Yaskawa INFORM job: pipe_bracket_cylinder_program.JBI

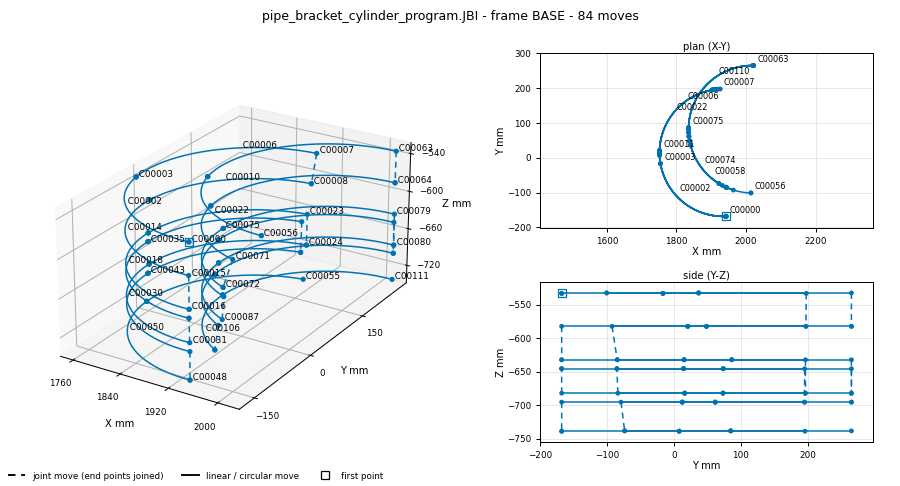
[picture p0: tool path of pipe_bracket_cylinder_program.JBI in frame BASE, 84 of 117 moves have a stored position in this frame; points joined in program order, loops and branches not executed]
/JOB
//NAME pipe_bracket_cylinder_program
//POS
///NPOS 112,0,112,0,0,0
///TOOL 0
///POSTYPE BASE
///RECTAN
///RCONF 0,0,0,0,0,0,0,0,0,0,0,0,0,0,0,0,0,0,0,0,0,0,0,0
C00000=1942.537957,-168.012753,-532.924500,-87.433791,-89.999999,5.000000
C00001=1942.537957,-168.012753,-532.924500,-87.433791,-89.999999,5.000000
C00002=1797.443653,-106.704534,-532.924500,-138.378261,-89.999999,5.000000
C00003=1753.930524,-16.502665,-532.924500,-170.116676,-89.999999,5.000000
C00004=1753.930524,-16.502665,-532.924500,-170.116676,-89.999999,5.000000
C00005=1753.930524,-16.502665,-532.924500,-170.116676,-89.999999,5.000000
C00006=1819.648743,157.692613,-532.924500,128.776952,-90.000000,5.000000
C00007=1925.886728,197.860249,-532.924500,92.645366,-90.000000,5.000000
C00008=1918.014662,197.326376,-582.169500,95.114199,-89.999999,5.000000
C00009=1918.014662,197.326376,-582.169500,95.114199,-89.999999,5.000000
C00010=1800.257643,139.658655,-582.169500,137.069440,-90.000000,5.000000
C00011=1751.301252,20.620145,-582.169500,175.000000,-89.999999,5.000000
C00012=1751.301252,20.620145,-582.169500,175.000000,-89.999999,5.000000
C00013=1751.301252,20.620145,-582.169500,175.000000,-89.999999,5.000000
C00014=1782.935371,-88.085662,-582.169500,-145.768544,-90.000000,5.000000
C00015=1941.730148,-168.047171,-582.169500,-87.686765,-90.000000,5.000000
C00016=1941.975553,-168.037093,-632.172000,-87.609919,-89.999999,5.000000
C00017=1941.975553,-168.037093,-632.172000,-87.609919,-89.999999,5.000000
C00018=1783.333373,-88.668199,-632.172000,-145.547804,-90.000000,5.000000
C00019=1751.212998,15.190866,-632.172000,175.000000,-90.000000,5.000000
C00020=1751.212998,15.190866,-632.172000,175.000000,-90.000000,5.000000
C00021=1751.212998,15.190866,-632.172000,175.000000,-90.000000,5.000000
C00022=1789.567117,127.073517,-632.172000,142.237662,-90.000000,5.000000
C00023=1912.126975,196.703354,-632.172000,96.966683,-90.000000,5.000000
C00024=1911.336404,196.605005,-682.155000,97.215941,-90.000000,5.000000
C00025=1911.336404,196.605005,-682.155000,97.215941,-90.000000,5.000000
C00026=1789.008166,126.348204,-682.155000,142.524163,-90.000000,5.000000
C00027=1751.215641,15.947385,-682.155000,175.000000,-90.000000,5.000000
C00028=1751.215641,15.947385,-682.155000,175.000000,-90.000000,5.000000
C00029=1751.215641,15.947385,-682.155000,175.000000,-90.000000,5.000000
C00030=1786.192815,-92.717556,-682.155000,-143.996770,-90.000000,5.000000
C00031=1942.358131,-168.020724,-682.155000,-87.490110,-90.000000,5.000000
C00032=1941.526633,-168.055278,-645.556460,-175.000000,-60.000000,92.249509
C00033=1941.526633,-168.055278,-645.556460,-175.000000,-60.000000,92.249509
C00034=1780.853143,-84.956813,-645.556460,175.000000,-60.000000,33.055529
C00035=1751.213846,14.313901,-645.556460,-175.000000,-60.000000,5.000000
C00036=1751.213846,14.313901,-645.556460,-175.000000,-60.000000,5.000000
C00037=1751.213846,14.313901,-645.556460,-175.000000,-60.000000,5.000000
C00038=1788.892614,126.197321,-645.556460,175.000000,-60.000000,-37.416375
C00039=1903.454355,195.432275,-645.556460,175.000000,-60.000000,-80.290608
C00040=1902.349178,195.239691,-695.542960,175.000000,-60.000000,-79.939613
C00041=1902.349178,195.239691,-695.542960,175.000000,-60.000000,-79.939613
C00042=1788.632983,125.857115,-695.542960,175.000000,-60.000000,-37.282477
C00043=1751.229898,12.427988,-695.542960,175.000000,-60.000000,5.000000
C00044=1751.229898,12.427988,-695.542960,175.000000,-60.000000,5.000000
C00045=1751.229898,12.427988,-695.542960,175.000000,-60.000000,5.000000
C00046=1782.456963,-87.379003,-695.542960,-175.000000,-60.000000,33.964456
C00047=1942.452445,-168.016565,-695.542960,175.000000,-60.000000,92.539427
C00048=1942.174784,-168.028668,-739.049960,-175.000000,-60.000000,92.452471
C00049=1942.174784,-168.028668,-739.049960,-175.000000,-60.000000,92.452471
C00050=1781.503320,-85.948835,-739.049960,175.000000,-60.000000,33.426633
C00051=1751.353161,7.761270,-739.049960,175.000000,-60.000000,5.000000
C00052=1751.353161,7.761270,-739.049960,175.000000,-60.000000,5.000000
C00053=1751.353161,7.761270,-739.049960,175.000000,-60.000000,5.000000
C00054=1784.506338,120.216512,-739.049960,175.000000,-60.000000,-35.095663
C00055=1906.907155,195.989172,-739.049960,-175.000000,-60.000000,-81.384886
C00056=2014.143483,-100.766826,-532.230000,-91.168935,-89.999999,5.000000
C00057=2014.143483,-100.766826,-532.230000,-91.168935,-89.999999,5.000000
C00058=1899.462167,-57.366095,-532.230000,-130.289001,-89.999999,5.000000
C00059=1840.487082,36.855691,-532.230000,-165.624641,-90.000000,5.000000
C00060=1840.487082,36.855691,-532.230000,-165.624641,-90.000000,5.000000
C00061=1840.487082,36.855691,-532.230000,-165.624641,-90.000000,5.000000
C00062=1900.582124,222.949781,-532.230000,129.831172,-90.000000,5.000000
C00063=2020.961875,265.420918,-532.230000,89.035494,-90.000000,5.000000
C00064=2020.657830,265.425784,-582.179500,89.130635,-89.999999,5.000000
C00065=2020.657830,265.425784,-582.179500,89.130635,-89.999999,5.000000
C00066=1885.350173,208.697868,-582.179500,136.361231,-89.999999,5.000000
C00067=1837.891489,48.564816,-582.179500,-169.377752,-90.000000,5.000000
C00068=1837.891489,48.564816,-582.179500,-169.377752,-90.000000,5.000000
C00069=1837.891489,48.564816,-582.179500,-169.377752,-90.000000,5.000000
C00070=1881.544380,-39.940562,-582.179500,-138.115094,-90.000000,5.000000
C00071=1963.739611,-92.618991,-582.179500,-107.196037,-90.000000,5.000000
C00072=1943.237520,-84.902532,-632.168500,-114.054049,-90.000000,5.000000
C00073=1943.237520,-84.902532,-632.168500,-114.054049,-90.000000,5.000000
C00074=1870.633273,-26.553727,-632.168500,-143.520535,-90.000000,5.000000
C00075=1834.799732,86.439422,-632.168500,175.000000,-90.000000,5.000000
C00076=1834.799732,86.439422,-632.168500,175.000000,-90.000000,5.000000
C00077=1834.799732,86.439422,-632.168500,175.000000,-90.000000,5.000000
C00078=1900.762842,223.100320,-632.168500,129.757582,-90.000000,5.000000
C00079=2021.100654,265.418529,-632.168500,88.992067,-89.999999,5.000000
C00080=2021.557535,265.409920,-682.170500,88.849094,-89.999999,5.000000
C00081=2021.557535,265.409920,-682.170500,88.849094,-89.999999,5.000000
C00082=1881.209361,204.207875,-682.170500,138.272336,-90.000000,5.000000
C00083=1834.977558,73.263237,-682.170500,-175.000000,-90.000000,5.000000
C00084=1834.977558,73.263237,-682.170500,-175.000000,-90.000000,5.000000
C00085=1834.977558,73.263237,-682.170500,-175.000000,-90.000000,5.000000
C00086=1869.380160,-24.838246,-682.170500,-144.185220,-89.999999,5.000000
C00087=1941.074160,-83.920016,-682.170500,-114.797455,-89.999999,5.000000
C00088=1944.487882,-85.455056,-645.550960,-175.000000,-60.000000,66.373654
C00089=1944.487882,-85.455056,-645.550960,-175.000000,-60.000000,66.373654
C00090=1872.022822,-28.408340,-645.550960,175.000000,-60.000000,37.204536
C00091=1834.960316,73.618385,-645.550960,175.000000,-60.000000,5.000000
C00092=1834.960316,73.618385,-645.550960,175.000000,-60.000000,5.000000
C00093=1834.960316,73.618385,-645.550960,175.000000,-60.000000,5.000000
C00094=1893.701616,216.912919,-645.550960,175.000000,-60.000000,-47.304641
C00095=2020.753432,265.424308,-645.550960,175.000000,-60.000000,-90.899280
C00096=2021.249895,265.415842,-695.548960,175.000000,-60.000000,-91.054635
C00097=2021.249895,265.415842,-695.548960,175.000000,-60.000000,-91.054635
C00098=1880.467269,203.370643,-695.548960,-175.000000,-60.000000,-41.377625
C00099=1835.921192,61.673045,-695.548960,175.000000,-60.000000,6.474015
C00100=1835.921192,61.673045,-695.548960,175.000000,-60.000000,6.474015
C00101=1835.921192,61.673045,-695.548960,175.000000,-60.000000,6.474015
C00102=1874.105058,-31.098868,-695.548960,175.000000,-60.000000,38.269005
C00103=1931.752214,-79.287259,-695.548960,-175.000000,-60.000000,61.945168
C00104=1922.138759,-73.784261,-738.575460,175.000000,-60.000000,58.478885
C00105=1922.138759,-73.784261,-738.575460,175.000000,-60.000000,58.478885
C00106=1874.782710,-31.952642,-738.575460,175.000000,-60.000000,38.610046
C00107=1834.769699,84.763058,-738.575460,-175.000000,-60.000000,-5.000000
C00108=1834.769699,84.763058,-738.575460,-175.000000,-60.000000,-5.000000
C00109=1834.769699,84.763058,-738.575460,-175.000000,-60.000000,-5.000000
C00110=1910.745399,230.838368,-738.575460,175.000000,-60.000000,-54.194979
C00111=2020.675033,265.425522,-738.575460,175.000000,-60.000000,-90.874748
///POSTYPE PULSE
///PULSE
EX00000=95232.0
EX00001=275456.0
///POSTYPE PULSE
///PULSE
EC00000=95232.0
EC00001=95232.0
EC00002=95232.0
EC00003=95232.0
EC00004=95232.0
EC00005=95232.0
EC00006=95232.0
EC00007=95232.0
EC00008=95232.0
EC00009=95232.0
EC00010=95232.0
EC00011=95232.0
EC00012=95232.0
EC00013=95232.0
EC00014=95232.0
EC00015=95232.0
EC00016=95232.0
EC00017=95232.0
EC00018=95232.0
EC00019=95232.0
EC00020=95232.0
EC00021=95232.0
EC00022=95232.0
EC00023=95232.0
EC00024=95232.0
EC00025=95232.0
EC00026=95232.0
EC00027=95232.0
EC00028=95232.0
EC00029=95232.0
EC00030=95232.0
EC00031=95232.0
EC00032=95232.0
EC00033=95232.0
EC00034=95232.0
EC00035=95232.0
EC00036=95232.0
EC00037=95232.0
EC00038=95232.0
EC00039=95232.0
EC00040=95232.0
EC00041=95232.0
EC00042=95232.0
EC00043=95232.0
EC00044=95232.0
EC00045=95232.0
EC00046=95232.0
EC00047=95232.0
EC00048=95232.0
EC00049=95232.0
EC00050=95232.0
EC00051=95232.0
EC00052=95232.0
EC00053=95232.0
EC00054=95232.0
EC00055=95232.0
EC00056=275456.0
EC00057=275456.0
EC00058=275456.0
EC00059=275456.0
EC00060=275456.0
EC00061=275456.0
EC00062=275456.0
EC00063=275456.0
EC00064=275456.0
EC00065=275456.0
EC00066=275456.0
EC00067=275456.0
EC00068=275456.0
EC00069=275456.0
EC00070=275456.0
EC00071=275456.0
EC00072=275456.0
EC00073=275456.0
EC00074=275456.0
EC00075=275456.0
EC00076=275456.0
EC00077=275456.0
EC00078=275456.0
EC00079=275456.0
EC00080=275456.0
EC00081=275456.0
EC00082=275456.0
EC00083=275456.0
EC00084=275456.0
EC00085=275456.0
EC00086=275456.0
EC00087=275456.0
EC00088=275456.0
EC00089=275456.0
EC00090=275456.0
EC00091=275456.0
EC00092=275456.0
EC00093=275456.0
EC00094=275456.0
EC00095=275456.0
EC00096=275456.0
EC00097=275456.0
EC00098=275456.0
EC00099=275456.0
EC00100=275456.0
EC00101=275456.0
EC00102=275456.0
EC00103=275456.0
EC00104=275456.0
EC00105=275456.0
EC00106=275456.0
EC00107=275456.0
EC00108=275456.0
EC00109=275456.0
EC00110=275456.0
EC00111=275456.0
//INST
///DATE 2023/08/16 18:21
///ATTR SC,RW,RJ
////FRAME BASE
///GROUP1 RB1,ST1
NOP
MOVJ P009 EX000 VJ=15.00
MOVJ C00000 EC00000 VJ=15.0
CALL JOB:SPYON
MOVC C00001 EC00001 V=150.0
MOVC C00002 EC00002 V=150.0
MOVC C00003 EC00003 V=150.0
MOVJ C00004 EC00004 VJ=15.0
MOVC C00005 EC00005 V=150.0
MOVC C00006 EC00006 V=150.0
MOVC C00007 EC00007 V=150.0
MOVJ C00008 EC00008 VJ=15.0
MOVC C00009 EC00009 V=150.0
MOVC C00010 EC00010 V=150.0
MOVC C00011 EC00011 V=150.0
MOVJ C00012 EC00012 VJ=15.0
MOVC C00013 EC00013 V=150.0
MOVC C00014 EC00014 V=150.0
MOVC C00015 EC00015 V=150.0
MOVJ C00016 EC00016 VJ=15.0
MOVC C00017 EC00017 V=150.0
MOVC C00018 EC00018 V=150.0
MOVC C00019 EC00019 V=150.0
MOVJ C00020 EC00020 VJ=15.0
MOVC C00021 EC00021 V=150.0
MOVC C00022 EC00022 V=150.0
MOVC C00023 EC00023 V=150.0
MOVJ C00024 EC00024 VJ=15.0
MOVC C00025 EC00025 V=150.0
MOVC C00026 EC00026 V=150.0
MOVC C00027 EC00027 V=150.0
MOVJ C00028 EC00028 VJ=15.0
MOVC C00029 EC00029 V=150.0
MOVC C00030 EC00030 V=150.0
MOVC C00031 EC00031 V=150.0
MOVJ C00032 EC00032 VJ=15.0
MOVC C00033 EC00033 V=150.0
MOVC C00034 EC00034 V=150.0
MOVC C00035 EC00035 V=150.0
MOVJ C00036 EC00036 VJ=15.0
MOVC C00037 EC00037 V=150.0
MOVC C00038 EC00038 V=150.0
MOVC C00039 EC00039 V=150.0
MOVJ C00040 EC00040 VJ=15.0
MOVC C00041 EC00041 V=150.0
MOVC C00042 EC00042 V=150.0
MOVC C00043 EC00043 V=150.0
MOVJ C00044 EC00044 VJ=15.0
MOVC C00045 EC00045 V=150.0
MOVC C00046 EC00046 V=150.0
MOVC C00047 EC00047 V=150.0
MOVJ C00048 EC00048 VJ=15.0
MOVC C00049 EC00049 V=150.0
MOVC C00050 EC00050 V=150.0
MOVC C00051 EC00051 V=150.0
MOVJ C00052 EC00052 VJ=15.0
MOVC C00053 EC00053 V=150.0
MOVC C00054 EC00054 V=150.0
MOVC C00055 EC00055 V=150.0
CALL JOB:SPYOF
MOVJ P009 VJ=15.00
MOVL P009 EX00000 V=150.0
MOVJ C00056 EC00056 VJ=15.0
CALL JOB:SPYON
MOVC C00057 EC00057 V=150.0
MOVC C00058 EC00058 V=150.0
MOVC C00059 EC00059 V=150.0
MOVJ C00060 EC00060 VJ=15.0
MOVC C00061 EC00061 V=150.0
MOVC C00062 EC00062 V=150.0
MOVC C00063 EC00063 V=150.0
MOVJ C00064 EC00064 VJ=15.0
MOVC C00065 EC00065 V=150.0
MOVC C00066 EC00066 V=150.0
MOVC C00067 EC00067 V=150.0
MOVJ C00068 EC00068 VJ=15.0
MOVC C00069 EC00069 V=150.0
MOVC C00070 EC00070 V=150.0
MOVC C00071 EC00071 V=150.0
MOVJ C00072 EC00072 VJ=15.0
MOVC C00073 EC00073 V=150.0
MOVC C00074 EC00074 V=150.0
MOVC C00075 EC00075 V=150.0
MOVJ C00076 EC00076 VJ=15.0
MOVC C00077 EC00077 V=150.0
MOVC C00078 EC00078 V=150.0
MOVC C00079 EC00079 V=150.0
MOVJ C00080 EC00080 VJ=15.0
MOVC C00081 EC00081 V=150.0
MOVC C00082 EC00082 V=150.0
MOVC C00083 EC00083 V=150.0
MOVJ C00084 EC00084 VJ=15.0
MOVC C00085 EC00085 V=150.0
MOVC C00086 EC00086 V=150.0
MOVC C00087 EC00087 V=150.0
MOVJ C00088 EC00088 VJ=15.0
MOVC C00089 EC00089 V=150.0
MOVC C00090 EC00090 V=150.0
MOVC C00091 EC00091 V=150.0
MOVJ C00092 EC00092 VJ=15.0
MOVC C00093 EC00093 V=150.0
MOVC C00094 EC00094 V=150.0
MOVC C00095 EC00095 V=150.0
MOVJ C00096 EC00096 VJ=15.0
MOVC C00097 EC00097 V=150.0
MOVC C00098 EC00098 V=150.0
MOVC C00099 EC00099 V=150.0
MOVJ C00100 EC00100 VJ=15.0
MOVC C00101 EC00101 V=150.0
MOVC C00102 EC00102 V=150.0
MOVC C00103 EC00103 V=150.0
MOVJ C00104 EC00104 VJ=15.0
MOVC C00105 EC00105 V=150.0
MOVC C00106 EC00106 V=150.0
MOVC C00107 EC00107 V=150.0
MOVJ C00108 EC00108 VJ=15.0
MOVC C00109 EC00109 V=150.0
MOVC C00110 EC00110 V=150.0
MOVC C00111 EC00111 V=150.0
CALL JOB:SPYOF
MOVJ P009 VJ=15.00
MOVL P009 EX00001 V=150.0
END
